// TIA Portal V18 export
FUNCTION_BLOCK "Drill"   // FB30, LAD
TITLE = Drill
{ S7_Optimized_Access := 'TRUE' }
// Written BY Kristopher Gimenez Feb 3,2023
// This block is used to control the TD Drill mode
// stored: AutoNumber false, MemoryReserve 100, SetENOAutomatically false
   VAR_INPUT
      DrillPSISet : Real;
      DisableThrottle : Bool;
   END_VAR
   VAR_OUTPUT
      FlowFwdmAOut : Real;
      FwdEnableP1 : Bool;
      TorquePSIOut : Real;
      FwdEnableP2 : Bool;
   END_VAR
   VAR
      PSinitialize : Bool := False;
      TorqLowLimitFtLbs { ExternalAccessible := 'False'; ExternalVisible := 'False'; ExternalWritable := 'False'} : Real;   // Above this value flow will be detroked
      TorqHighLimitFtLbs : Real;
      TorqLimiting : Bool;   // Bit to indicate torq limiting
      TorqLimitTrig : Bool;   // Bit used for positive trigger transition on Torq Limiting
      LimitFlowmAOut : Real;   // Calculated limited output value for flow
      TorqLimit_TON { S7_SetPoint := 'True'} : TON_TIME;
      TorqLimit_SlewDec { S7_SetPoint := 'True'} : "SlewDec";
      Torq_Limit_SlewInc { S7_SetPoint := 'True'} : "SlewInc";
   END_VAR
   VAR_TEMP
      PSIsetHIgh : Real;
      PSIsetLow : Real;
      PSIcheck : Real;
      PSiRange : Real;
      PSIadjustRange : Real;
      PSIadjustval : Real;
      PsiPos : Bool;
      PSIinitial : Bool;
      PSIAdjust : Bool;
      FlowmAOutTemp : Real;
      TempPSI : Real;
      tempReal : Real;
   END_VAR
   VAR_TEMP   // added for the SCL form of the ladder/FBD networks
      _w1 : Bool;
      _w2 : Bool;
      _w3 : Bool;
   END_VAR
BEGIN

REGION Network 1: Speed Setpoint
   // If throttle not disable get speed setpoint
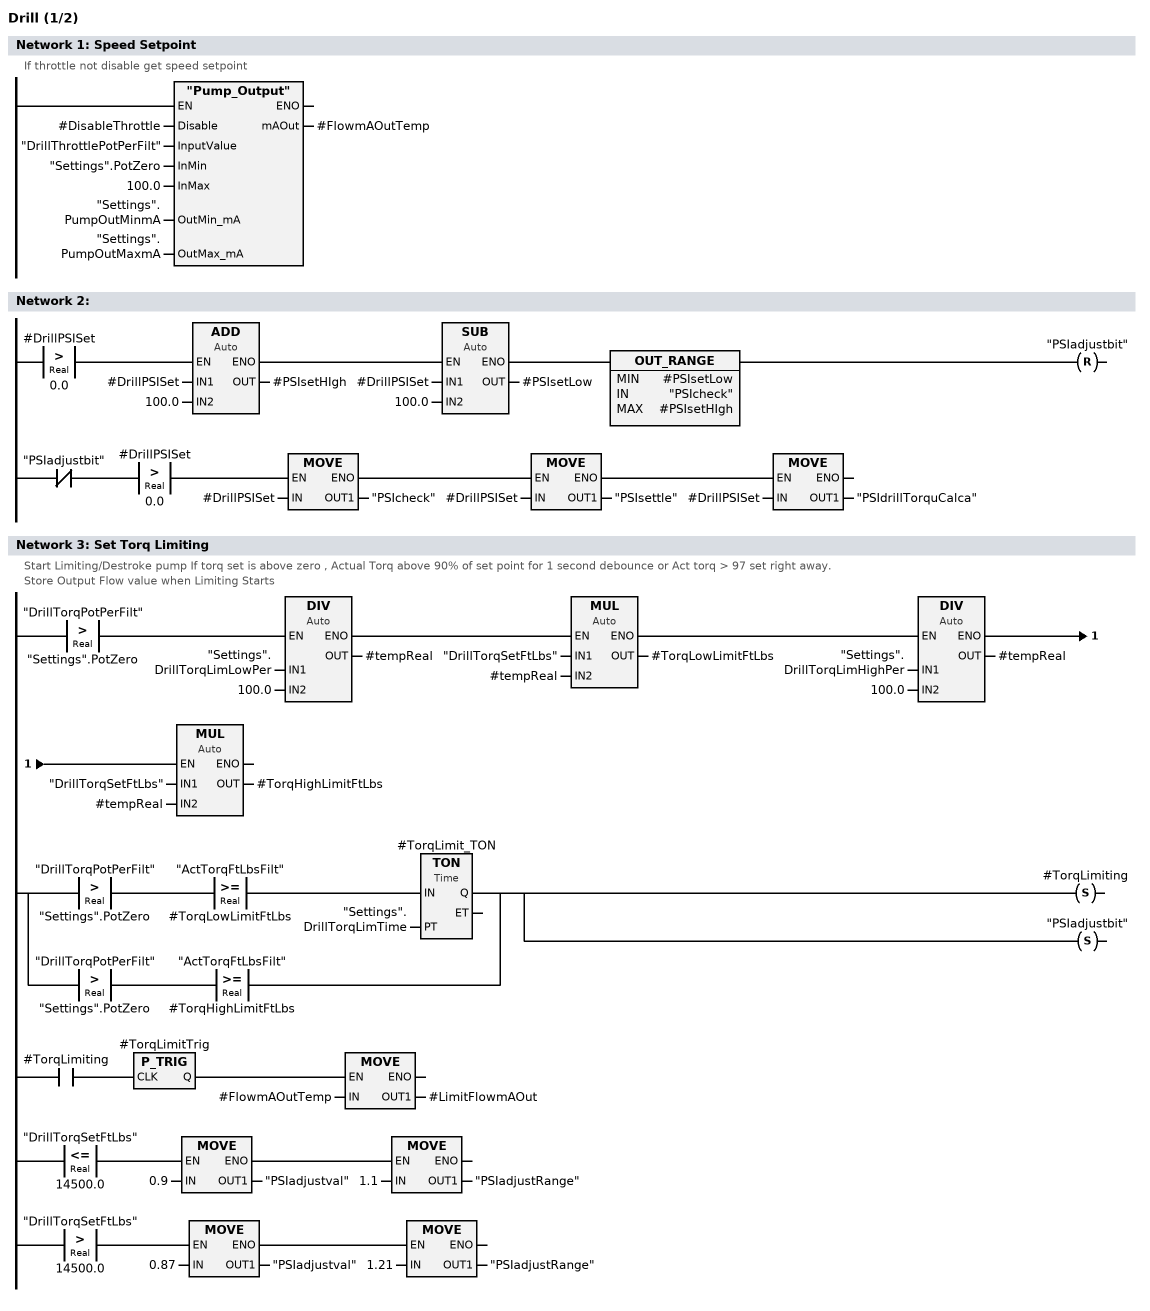
   RUNG wire#powerrail
      "Pump_Output"(Disable := #DisableThrottle, InputValue := "DrillThrottlePotPerFilt", InMin := "Settings".PotZero, InMax := 100.0, OutMin_mA := "Settings".PumpOutMinmA, OutMax_mA := "Settings".PumpOutMaxmA, mAOut => #FlowmAOutTemp)
   END_RUNG
   // the same network as SCL:
   "Pump_Output"(Disable := #DisableThrottle,
                 InputValue := "DrillThrottlePotPerFilt",
                 InMin := "Settings".PotZero,
                 InMax := 100.0,
                 OutMin_mA := "Settings".PumpOutMinmA,
                 OutMax_mA := "Settings".PumpOutMaxmA,
                 mAOut => #FlowmAOutTemp);
END_REGION

REGION Network 2
   #_w1 := #DrillPSISet > 0.0;
   IF #_w1 THEN
       #PSIsetHIgh := #DrillPSISet + 100.0;
       #PSIsetLow := #DrillPSISet - 100.0;
   END_IF;
   IF #_w1 AND (("PSIcheck" < #PSIsetLow) OR ("PSIcheck" > #PSIsetHIgh)) THEN
       "PSIadjustbit" := FALSE;
   END_IF;
   IF NOT "PSIadjustbit" AND (#DrillPSISet > 0.0) THEN
       "PSIcheck" := #DrillPSISet;
       "PSIsettle" := #DrillPSISet;
       "PSIdrillTorquCalca" := #DrillPSISet;
   END_IF;
END_REGION

REGION Network 3: Set Torq Limiting
   // Start Limiting/Destroke pump If torq set is above zero , Actual Torq above 90% of set point for 1 second debounce or Act torq > 97 set right away. 
   // Store Output Flow value when Limiting Starts
   RUNG wire#powerrail
      { S7_Templates := "SrcType := Real" } GT_Contact(in1 := "DrillTorqPotPerFilt", in2 := "Settings".PotZero)
      Div(in1 := "Settings".DrillTorqLimLowPer, in2 := 100.0, out => #tempReal)
      Mul(in1 := "DrillTorqSetFtLbs", in2 := #tempReal, out => #TorqLowLimitFtLbs)
      Div(in1 := "Settings".DrillTorqLimHighPer, in2 := 100.0, out => #tempReal)
      Mul(in1 := "DrillTorqSetFtLbs", in2 := #tempReal, out => #TorqHighLimitFtLbs)
   END_RUNG
   RUNG wire#powerrail
      { S7_Templates := "SrcType := Real" } GT_Contact(in1 := "DrillTorqPotPerFilt", in2 := "Settings".PotZero)
      { S7_Templates := "SrcType := Real" } GE_Contact(in1 := "ActTorqFtLbsFilt", in2 := #TorqLowLimitFtLbs)
      { S7_Templates := "time_type := Time" } #TorqLimit_TON.TON(pt := "Settings".DrillTorqLimTime, et =>)
      wire#w1
      S_Coil( #TorqLimiting )
   END_RUNG
   RUNG wire#powerrail
      { S7_Templates := "SrcType := Real" } GT_Contact(in1 := "DrillTorqPotPerFilt", in2 := "Settings".PotZero)
      { S7_Templates := "SrcType := Real" } GE_Contact(in1 := "ActTorqFtLbsFilt", in2 := #TorqHighLimitFtLbs)
   END_RUNG wire#w1
   RUNG wire#w1
      S_Coil( "PSIadjustbit" )
   END_RUNG
   RUNG wire#powerrail
      Contact( #TorqLimiting )
      P_Trig( #TorqLimitTrig )
      Move(in := #FlowmAOutTemp, out1 => #LimitFlowmAOut)
   END_RUNG
   RUNG wire#powerrail
      { S7_Templates := "SrcType := Real" } LE_Contact(in1 := "DrillTorqSetFtLbs", in2 := 14500.0)
      Move(in := 0.9, out1 => "PSIadjustval")
      Move(in := 1.1, out1 => "PSIadjustRange")
   END_RUNG
   RUNG wire#powerrail
      { S7_Templates := "SrcType := Real" } GT_Contact(in1 := "DrillTorqSetFtLbs", in2 := 14500.0)
      Move(in := 0.87, out1 => "PSIadjustval")
      Move(in := 1.21, out1 => "PSIadjustRange")
   END_RUNG
   // the same network as SCL:
   IF "DrillTorqPotPerFilt" > "Settings".PotZero THEN
       #tempReal := "Settings".DrillTorqLimLowPer / 100.0;
       #TorqLowLimitFtLbs := "DrillTorqSetFtLbs" * #tempReal;
       #tempReal := "Settings".DrillTorqLimHighPer / 100.0;
       #TorqHighLimitFtLbs := "DrillTorqSetFtLbs" * #tempReal;
   END_IF;
   #TorqLimit_TON(IN := ("DrillTorqPotPerFilt" > "Settings".PotZero) AND ("ActTorqFtLbsFilt" >= #TorqLowLimitFtLbs),   // TON
                  PT := "Settings".DrillTorqLimTime);
   IF #TorqLimit_TON.Q OR (("DrillTorqPotPerFilt" > "Settings".PotZero) AND ("ActTorqFtLbsFilt" >= #TorqHighLimitFtLbs)) THEN
       #TorqLimiting := TRUE;
       "PSIadjustbit" := TRUE;
   END_IF;
   #_w1 := #TorqLimiting AND NOT #TorqLimitTrig;   // rising edge
   #TorqLimitTrig := #TorqLimiting;
   IF #_w1 THEN #LimitFlowmAOut := #FlowmAOutTemp; END_IF;
   IF "DrillTorqSetFtLbs" <= 14500.0 THEN
       "PSIadjustval" := 0.9;
       "PSIadjustRange" := 1.1;
   END_IF;
   IF "DrillTorqSetFtLbs" > 14500.0 THEN
       "PSIadjustval" := 0.87;
       "PSIadjustRange" := 1.21;
   END_IF;
END_REGION

REGION Network 4: Flow Control in Torq Limit
   // If torq limiting-
   // in High torq  destroke the ouput. 
   // - if low torq increase stroke back to setpoint
   // -Otherwise hold.  
   // Slew rate are mA/sec. TON increment set to 10ms so unput Slew rate divided by 100
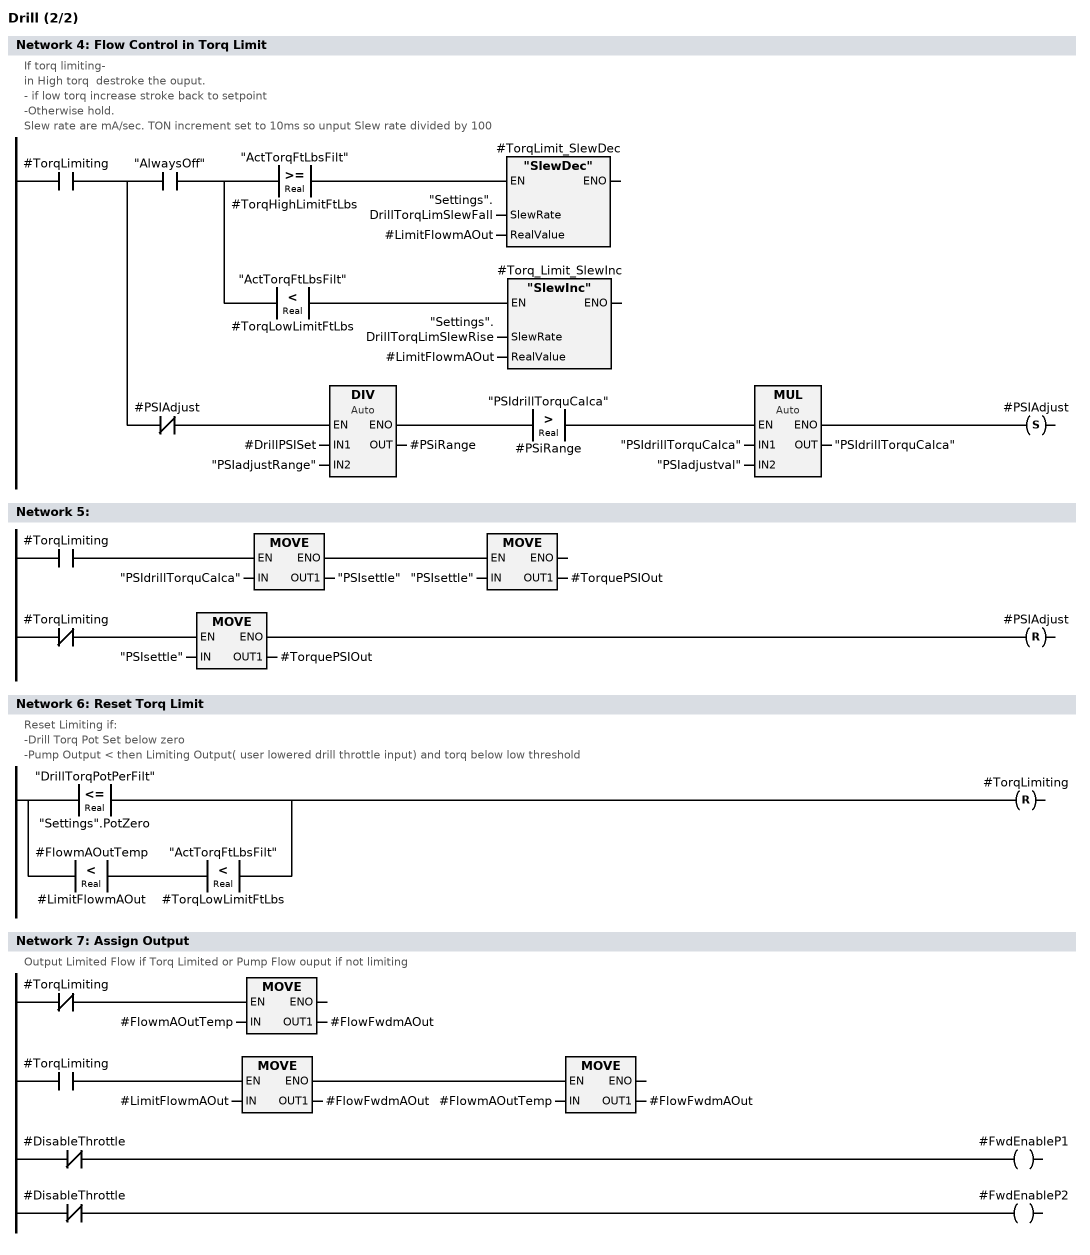
   RUNG wire#powerrail
      Contact( #TorqLimiting )
      wire#w1
      Contact( "AlwaysOff" )
      wire#w2
      { S7_Templates := "SrcType := Real" } GE_Contact(in1 := "ActTorqFtLbsFilt", in2 := #TorqHighLimitFtLbs)
      #TorqLimit_SlewDec(SlewRate := "Settings".DrillTorqLimSlewFall, RealValue := #LimitFlowmAOut)
   END_RUNG
   RUNG wire#w2
      { S7_Templates := "SrcType := Real" } LT_Contact(in1 := "ActTorqFtLbsFilt", in2 := #TorqLowLimitFtLbs)
      #Torq_Limit_SlewInc(SlewRate := "Settings".DrillTorqLimSlewRise, RealValue := #LimitFlowmAOut)
   END_RUNG
   RUNG wire#w1
      I_Contact( #PSIAdjust )
      Div(in1 := #DrillPSISet, in2 := "PSIadjustRange", out => #PSiRange)
      { S7_Templates := "SrcType := Real" } GT_Contact(in1 := "PSIdrillTorquCalca", in2 := #PSiRange)
      Mul(in1 := "PSIdrillTorquCalca", in2 := "PSIadjustval", out => "PSIdrillTorquCalca")
      S_Coil( #PSIAdjust )
   END_RUNG
   // the same network as SCL:
   #_w1 := #TorqLimiting AND "AlwaysOff";
   IF #_w1 AND ("ActTorqFtLbsFilt" >= #TorqHighLimitFtLbs) THEN
       #TorqLimit_SlewDec(SlewRate := "Settings".DrillTorqLimSlewFall, RealValue := #LimitFlowmAOut);   // "SlewDec"
   END_IF;
   IF #_w1 AND ("ActTorqFtLbsFilt" < #TorqLowLimitFtLbs) THEN
       #Torq_Limit_SlewInc(SlewRate := "Settings".DrillTorqLimSlewRise, RealValue := #LimitFlowmAOut);   // "SlewInc"
   END_IF;
   #_w2 := #TorqLimiting AND NOT #PSIAdjust;
   IF #_w2 THEN #PSiRange := #DrillPSISet / "PSIadjustRange"; END_IF;
   #_w3 := #_w2 AND ("PSIdrillTorquCalca" > #PSiRange);
   IF #_w3 THEN
       "PSIdrillTorquCalca" := "PSIdrillTorquCalca" * "PSIadjustval";
       #PSIAdjust := TRUE;
   END_IF;
END_REGION

REGION Network 5
   RUNG wire#powerrail
      Contact( #TorqLimiting )
      Move(in := "PSIdrillTorquCalca", out1 => "PSIsettle")
      Move(in := "PSIsettle", out1 => #TorquePSIOut)
   END_RUNG
   RUNG wire#powerrail
      I_Contact( #TorqLimiting )
      Move(in := "PSIsettle", out1 => #TorquePSIOut)
      R_Coil( #PSIAdjust )
   END_RUNG
   // the same network as SCL:
   IF #TorqLimiting THEN
       "PSIsettle" := "PSIdrillTorquCalca";
       #TorquePSIOut := "PSIsettle";
   END_IF;
   IF NOT #TorqLimiting THEN
       #TorquePSIOut := "PSIsettle";
       #PSIAdjust := FALSE;
   END_IF;
END_REGION

REGION Network 6: Reset Torq Limit
   // Reset Limiting if:
   // -Drill Torq Pot Set below zero
   //  -Pump Output < then Limiting Output( user lowered drill throttle input) and torq below low threshold
   RUNG wire#powerrail
      { S7_Templates := "SrcType := Real" } LE_Contact(in1 := "DrillTorqPotPerFilt", in2 := "Settings".PotZero)
      wire#w1
      R_Coil( #TorqLimiting )
   END_RUNG
   RUNG wire#powerrail
      { S7_Templates := "SrcType := Real" } LT_Contact(in1 := #FlowmAOutTemp, in2 := #LimitFlowmAOut)
      { S7_Templates := "SrcType := Real" } LT_Contact(in1 := "ActTorqFtLbsFilt", in2 := #TorqLowLimitFtLbs)
   END_RUNG wire#w1
   // the same network as SCL:
   IF ("DrillTorqPotPerFilt" <= "Settings".PotZero) OR ((#FlowmAOutTemp < #LimitFlowmAOut) AND ("ActTorqFtLbsFilt" < #TorqLowLimitFtLbs)) THEN
       #TorqLimiting := FALSE;
   END_IF;
END_REGION

REGION Network 7: Assign Output
   // Output Limited Flow if Torq Limited or Pump Flow ouput if not limiting
   RUNG wire#powerrail
      I_Contact( #TorqLimiting )
      Move(in := #FlowmAOutTemp, out1 => #FlowFwdmAOut)
   END_RUNG
   RUNG wire#powerrail
      Contact( #TorqLimiting )
      Move(in := #LimitFlowmAOut, out1 => #FlowFwdmAOut)
      Move(in := #FlowmAOutTemp, out1 => #FlowFwdmAOut)
   END_RUNG
   RUNG wire#powerrail
      I_Contact( #DisableThrottle )
      Coil( #FwdEnableP1 )
   END_RUNG
   RUNG wire#powerrail
      I_Contact( #DisableThrottle )
      Coil( #FwdEnableP2 )
   END_RUNG
   // the same network as SCL:
   IF NOT #TorqLimiting THEN #FlowFwdmAOut := #FlowmAOutTemp; END_IF;
   IF #TorqLimiting THEN
       #FlowFwdmAOut := #LimitFlowmAOut;
       #FlowFwdmAOut := #FlowmAOutTemp;
   END_IF;
   #FwdEnableP1 := NOT #DisableThrottle;
   #FwdEnableP2 := NOT #DisableThrottle;
END_REGION
END_FUNCTION_BLOCK
